FUNCTION_BLOCK FB_CommandChangeDiagnostics EXTENDS FB_CommandChange IMPLEMENTS ITF_CommandChange
VAR

END_VAR

(*			
	RafalOS
	Rafał Osajda		03.11.2025		TC 4024.66
	Test czy można zmienić stan lub tryb i zwraca czy można i uruchamia zmianę
*)
METHOD PUBLIC Execute : BOOL
VAR_INPUT
	iNumberOfCommand	: INT;
END_VAR
IF (THIS^.itfSaMController.IsModeEnebles (eMode := E_BaseMachineMode.Diagnostics)) THEN
	IF (THIS^.itfSaMController.IsPossibleExitActiveState ()) THEN
		IF (THIS^.itfSaMController.IsPossibleExitState (eMode := E_BaseMachineMode.Diagnostics)) THEN
			THIS^.itfSaMController.ChangeModeTo (eNewMode := E_BaseMachineMode.Diagnostics);
		ELSE
			THIS^.EventSetActive (iNumber := 3);	//brak możlwiosći wejście do trybu w tym stanie 
		END_IF
	ELSE
		THIS^.EventSetActive (iNumber := 2);	//brak możliwości wyjścia w tym stanie z tego trybu
	END_IF
ELSE
	THIS^.EventSetActive (iNumber := 1);	//tryb docelowy wylaczony
END_IF
END_METHOD

METHOD FB_init : BOOL
VAR_INPUT
	bInitRetains : BOOL; // if TRUE, the retain variables are initialized (warm start / cold start)
	bInCopyCode : BOOL;  // if TRUE, the instance afterwards gets moved into the copy code (online change)
END_VAR
THIS^.SetText (eLocation := E_BaseLocation.pl, wsDescription := "Command change mode - Diagnostics");
THIS^.SetText (eLocation := E_BaseLocation.en, wsDescription := "Command change mode - Diagnostics");
THIS^.SetText (eLocation := E_BaseLocation.de, wsDescription := "Command change mode - Diagnostics");
THIS^.SetName (stName := THIS^.GetTexts ());
END_METHOD

END_FUNCTION_BLOCK

(* stored: Version 1.1.0.1
   POU FB_CommandChangeDiagnostics: Id {ed383c6a-d475-0169-01d9-89d0a8244ba2}, SpecialFunc None
   Method Execute: Id {ff40543e-f6c7-0440-0ff0-634f85cf471f}
   Method FB_init: Id {43ad3b51-3956-02ef-381f-d2b600fa14b2} *)
